# B&R Automation Studio project GroupProjectBR (part 3)

```iecst
			httpDecodeBase64_0();	// call FUB

			IF NOT(httpDecodeBase64_0.destLen=0) THEN
				Base64srcLen := httpDecodeBase64_0.destLen;
				httpDecodeBase64_0.enable := FALSE;
				ImageProcess := 0;
			END_IF;
	END_CASE;

END_PROGRAM

PROGRAM _EXIT
	(* Insert code here *)

END_PROGRAM
```

### Program Logical/Programs/Alarms (IEC)

#### Variables.var
```iecst
VAR
	test_alarm : BOOL;
	MpAlarmXCore_0 : MpAlarmXCore;
	pendingAlarms : BOOL;
	enableRedIcon : BOOL;
	enableYellowIcon : BOOL;
	redIconTimer : TON;
	timerCycle : BOOL;
	MpAlarmXHistory_0 : MpAlarmXHistory;
	MpUserXConfigType_0 : MpUserXConfigType;
	MpUserXConfig_0 : MpUserXConfig;
	isAcknowledged : BOOL;
	IsSemiAutoMode : BOOL;
	IsManualMode : BOOL;
END_VAR
```

#### Main.st
```iecst
PROGRAM _INIT
	(* Insert code here *)

END_PROGRAM

PROGRAM _CYCLIC
	(* Insert code here *)
	MpAlarmXCore_0.Enable := TRUE;
	MpAlarmXCore_0.MpLink := ADR(gAlarmXCore);
	MpAlarmXCore_0();

	MpAlarmXHistory_0.Enable := TRUE;
	MpAlarmXHistory_0.MpLink := ADR(gAlarmXHistory);
	MpAlarmXHistory_0();

	MpUserXConfig_0.Enable := TRUE;
	MpUserXConfig_0.Configuration := ADR(MpUserXConfigType_0);
	MpUserXConfig_0();

	redIconTimer.PT := T#500ms;
	redIconTimer();

	// HARDWARE ALARM DETECTION
	IF NOT ModuleOkActuators OR NOT ModuleOkCamera OR NOT ModuleOkEncoder OR NOT ModuleOkInverter OR NOT ModuleOkPLC_PLK OR NOT ModuleOkPneu_X67BC OR NOT ModuleOkScale THEN
		gAlarmHardware := TRUE;
	ELSE
		gAlarmHardware := FALSE;
	END_IF;

	//isAcknowledged := MpAlarmXCheckState(gAlarmXCore, 'test_alarm', mpALARMX_STATE_ACKNOWLEDGED);
	IF (MpAlarmXCheckState(gAlarmXCore, 'Unrecognized object', mpALARMX_STATE_ACKNOWLEDGED) AND
		MpAlarmXCheckState(gAlarmXCore, 'Left box is full', mpALARMX_STATE_ACKNOWLEDGED) AND
		MpAlarmXCheckState(gAlarmXCore, 'Hardware error', mpALARMX_STATE_ACKNOWLEDGED) AND
		MpAlarmXCheckState(gAlarmXCore, 'Motor error', mpALARMX_STATE_ACKNOWLEDGED) AND
		MpAlarmXCheckState(gAlarmXCore, 'Right box is full', mpALARMX_STATE_ACKNOWLEDGED)) THEN
		isAcknowledged := TRUE;
	ELSE
		isAcknowledged := FALSE;
	END_IF;

	IF (MpAlarmXCore_0.PendingAlarms > 0) THEN
		pendingAlarms := TRUE;
	ELSE
		pendingAlarms := FALSE;
	END_IF;

	IF (MpAlarmXCore_0.ActiveAlarms = 0 AND MpAlarmXCore_0.PendingAlarms > 0) THEN
		enableYellowIcon := TRUE;
	ELSE
		enableYellowIcon := FALSE;
	END_IF;

	IF (MpAlarmXCore_0.ActiveAlarms > 0) THEN
		gAlarmExist := TRUE;
		IF (NOT(isAcknowledged)) THEN
			//blinking
			IF (redIconTimer.IN = FALSE) THEN
				redIconTimer.IN := TRUE;
			ELSIF (redIconTimer.Q) THEN
				timerCycle := NOT timerCycle;
				redIconTimer.IN := FALSE;
			END_IF;
			enableRedIcon := timerCycle;
		ELSE
			//static
			enableRedIcon := TRUE;
		END_IF;
	ELSE
		gAlarmExist := FALSE;
		enableRedIcon := FALSE;
	END_IF;

END_PROGRAM

PROGRAM _EXIT
	(* Insert code here *)

END_PROGRAM
```

### Program Logical/Programs/PustyProgram

#### Main.st
```iecst
PROGRAM _INIT

END_PROGRAM

PROGRAM _CYCLIC

END_PROGRAM

PROGRAM _EXIT
	(* Insert code here *)

END_PROGRAM
```

### Program Logical/Programs/SemiAuto

#### Variables.var
```iecst
VAR
	Approval : BOOL;
	ActuatorByte : INT := 2#0000000000000000;
	ActuatorNotPushing : BOOL;
	ActuatorNotSorting : BOOL;
	ActuatorPushing : BOOL := FALSE;
	ActuatorSorting : BOOL := FALSE;
END_VAR
VAR CONSTANT
	ACTUATOR_BYTE_NOT_ACTIV : USINT := 2#0000000000000000;
	ACTUATOR_BYTE_PUSH : INT := 2#0000000000000100;
	ACTUATOR_BYTE_SORT : INT := 2#0000000000000001;
END_VAR
VAR
	AddToLeft : BOOL;
	AddToRight : BOOL;
	CTU_QuantityLeft : CTU;
	CTU_QuantityRight : CTU;
	CTU_Reset_Left : BOOL := FALSE;
	CTU_Reset_Right : BOOL;
	IsEnglishSelected : BOOL := TRUE;
	ItemDetected : BOOL := FALSE;
	ItemWeight : USINT;
	ItemWeightMeasured : USINT;
	MotorHome : BOOL;
	MotorInPosition : BOOL;
	MotorMoveAbsolute : BOOL := FALSE;
	MotorMoveDone : BOOL;
	MotorPos : LREAL;
	MotorPower : BOOL := FALSE;
	MotorReqAcc : UINT := 700;
	MotorReqDec : UINT := 700;
	MotorReqPosition : UINT := 0;
	MotorReqVel : {REDUND_UNREPLICABLE} UINT := 300;
	MotorResetError : BOOL := FALSE;
	MotorVel : REAL;
END_VAR
VAR CONSTANT
	MOTOR_DIST_LEFT : UINT := 90;
	MOTOR_DIST_RIGHT : UINT := 320;
END_VAR
VAR
	QuantityLeftStorage : UINT;
	QuantityRightStorage : UINT;
END_VAR
VAR CONSTANT
	RESET_ITEM_MEM_WEIGHT : USINT := 0;
END_VAR
VAR
	Start : BOOL := FALSE;
	State : ProgramStatesEnum := STOP;
	Stop : BOOL := FALSE;
	StringRecognisedModel : STRING[80];
	StringState : STRING[80];
	TimerActuatorOut : BOOL;
	TimerAfterDetect : BOOL;
	TimerCameraPicDone : BOOL;
	TimerTonActuator : TON;
	TimerTonActuatorIn : BOOL := FALSE;
	TimerTonCamera : TON;
	TimerTonDetect : TON;
END_VAR
VAR CONSTANT
	TIME_TON_ACTUATOR : TIME := T#500MS;
	TIME_TON_CAMERA : TIME := T#4S;
END_VAR
VAR
	TIME_TON_DETECT : TIME := T#2S;
	SemiAutoModeSelected : BOOL;
END_VAR
```

#### Main.st
```iecst
// ALREADY WORKING
PROGRAM _INIT
	// NEED ONLY FOR WATCH
	gAxis_1;
	gMotorBeltParType;
	gMotorBeltAxisBasic;
END_PROGRAM

PROGRAM _CYCLIC
	//CODE WORKS ONLY WHEN MANUAL MODE IS OFF
	SemiAutoModeSelected := (gMode=2);
	IF  SemiAutoModeSelected THEN
		// MOTOR MANAGEMENT
		gMotorBeltAxisBasic.Enable 		:= TRUE;
		gMotorBeltAxisBasic.MpLink 		:= ADR(gAxis_1);
		gMotorBeltAxisBasic.Parameters 	:= ADR(gMotorBeltParType);
		MotorMoveDone 					:= gMotorBeltAxisBasic.MoveDone;
		gMotorBeltAxisBasic.Power 		:= MotorPower;
		gMotorBeltAxisBasic.Home 		:= MotorHome;

		// IN STATE STOP VALUES DOESN'T FLUCTUATE
		IF gMotorBeltAxisBasic.Velocity > 15 THEN
			MotorVel := gMotorBeltAxisBasic.Velocity;
		ELSE
			MotorVel := 0;
		END_IF;
		IF gMotorBeltAxisBasic.Position > 5 THEN
			MotorPos := gMotorBeltAxisBasic.Position;
		ELSE
			MotorPos := 0;
		END_IF;

		// ASSIGNING MOTION PARAMETERS
		gMotorBeltParType.Acceleration 	:= MotorReqAcc;
		gMotorBeltParType.Deceleration 	:= MotorReqDec;
		gMotorBeltParType.Velocity 		:= MotorReqVel;
		gMotorBeltParType.Position 		:= MotorReqPosition;

		gMotorBeltAxisBasic();

		// ASSIGNING GLOBAL VARIABLES TO LOCAL VARIABLES
		gActuatorByte					 := ActuatorByte;
		gMotorBeltAxisBasic.Power 		 := MotorPower;
		gMotorBeltAxisBasic.MoveAbsolute := MotorMoveAbsolute;
		gMotorBeltAxisBasic.ErrorReset	 := MotorResetError;
		gStopState 						 := (State = 0);

		// ASSIGNING LOCAL VARIABLES TO GLOBAL VARIABLES
		MotorInPosition 				 := gMotorBeltAxisBasic.InPosition;
		ItemWeight 						 := gInWeightMeasure;

		// ITEM DETECTION CONDITION
		ItemDetected := (ItemWeight > 1);
		gWeightDetected := ItemDetected;

		// TIMERS
		// actuator
		TimerTonActuator(IN := TimerTonActuatorIn, PT := TIME_TON_ACTUATOR);
		TimerActuatorOut := TimerTonActuator.Q;
		// camera
		TimerTonCamera(IN := gImageAcq , PT := TIME_TON_CAMERA);
		TimerCameraPicDone := TimerTonCamera.Q;
		// delay after detection
		TimerTonDetect.IN := ItemDetected;
		TimerTonDetect.PT := TIME_TON_DETECT;
		TimerAfterDetect := TimerTonDetect.Q;
		TimerTonDetect();

		// COUNTERS - PRZENIESIONY NA SZYBKO DO AUTO

	END_IF;

	// ALARM OR STOP OR MANUAL TURNED ON
	IF	gAlarmHardware THEN	//ALARM
		IF NOT (State = ERROR) THEN
			State := ERROR;
		END_IF;
	ELSIF Stop OR NOT SemiAutoModeSelected OR gAlarmExist THEN
		Stop := FALSE;
		State := STOP;
	END_IF;

	// PROGRAM AUTO
	CASE State OF
		STOP:
			IF SemiAutoModeSelected THEN
				MotorPower 		  := FALSE;
				MotorMoveAbsolute := FALSE;
				MotorHome 		  := FALSE;
				MotorResetError   := FALSE;
			END_IF;
			MotorPos := 0;
			MotorVel := 0;
			StringState := 'Stop';
			TimerTonActuatorIn 	  := FALSE;
			ActuatorSorting 	  := FALSE;
			ActuatorPushing  	  := FALSE;
			IF Start THEN
				State := INIT;
			END_IF;

		INIT:
			StringState 		:= 'Inicjalizacja';
			ItemWeightMeasured 	:= RESET_ITEM_MEM_WEIGHT;
			gAddToRight 		:= FALSE;
			gAddToLeft 			:= FALSE;
			TimerTonActuatorIn 	:= FALSE;
			ActuatorSorting 	:= FALSE;
			ActuatorPushing 	:= FALSE;
			MotorMoveAbsolute 	:= FALSE;
			MotorPower 			:= TRUE;
			MotorHome 			:= TRUE;
			gPicNotRecognised	:= FALSE;
			State 				:= START;

		START:
			StringState 		:= 'Gotowy do startu';
			IF (ItemDetected AND Approval) THEN
				Approval := 0;
				State := DETECTION;
			END_IF;

		DETECTION:
			MotorHome 	:= FALSE;
			StringState := 'Wykrycie detalu';
			IF TimerAfterDetect THEN
				ItemWeightMeasured := ItemWeight;
				State := CATEGORIZATION;
			END_IF;

		CATEGORIZATION:
			StringState := 'Kategoryzacja detalu';
			IF gSorting.SortChoice = WEIGHT THEN
				State := DROP;
			ELSIF gSorting.SortChoice = OPTIC THEN
				State := TAKE_PICT_CAMERA;
			END_IF;

		TAKE_PICT_CAMERA:
			StringState := 'Robienie zdjecia';
			gImageAcq 	:= TRUE;
			IF TimerCameraPicDone AND Approval THEN
				StringState := 'Zdjecie zrobione';
				gDisplayImg := TRUE;
				Approval := 0;
				IF gSorting.RecognisedModel = 0 THEN 						//0
					gImageAcq 			  := FALSE;
					StringRecognisedModel := 'Unrecognised';
					State 				  := UNRECOGNISED_PIC;
				ELSE
					State 				  := DROP;
				END_IF;
			END_IF;

		DROP:
			StringState := 'Dozowanie detalu';
			ActuatorPushing := TRUE;
			IF TimerActuatorOut THEN
				ActuatorPushing := FALSE;
				IF gSorting.SortChoice = OPTIC THEN
					gSortChoiceView := TRUE;
					State := SORT_OPTIC;
				ELSIF gSorting.SortChoice = WEIGHT THEN
					gSortChoiceView := FALSE;
					State := SORT_WEIGHT;
				END_IF;
			END_IF;

		// ABOVE 1 TO ItemWeightChoosen ITEM FALL INTO THE LEFT, EQUAL AND ABOVE ItemWeightChoosen INTO THE RIGHT
		SORT_WEIGHT:
			StringState := 'Sortowanie wagowe';
			IF ItemWeightMeasured > 1 AND ItemWeightMeasured < gSorting.ItemWeightChoosen AND Approval THEN
				IF gSorting.SortLeftMin THEN
					Approval := 0;
					State := GO_STORAGE_LEFT;
				ELSE
					Approval := 0;
					State := GO_STORAGE_RIGHT;
				END_IF;
			ELSIF ItemWeightMeasured >= gSorting.ItemWeightChoosen AND Approval THEN
				IF gSorting.SortLeftMin THEN
					Approval := 0;
					State := GO_STORAGE_RIGHT;
				ELSE
					Approval := 0;
					State := GO_STORAGE_LEFT;
				END_IF;
			END_IF;

		SORT_OPTIC:
			StringState := 'Sortowanie optyczne';
			IF gSorting.RecognisedModel = 1 THEN
				gImageAcq 			  := FALSE;
				StringRecognisedModel := 'B&R';					//1
				IF gSorting.SortLeftBR AND Approval THEN
					Approval := 0;
					State := GO_STORAGE_LEFT;
				ELSE
					IF Approval THEN
						Approval := 0;
						State := GO_STORAGE_RIGHT;
					END_IF;
				END_IF;

			ELSIF gSorting.RecognisedModel = 2 THEN						//2
				gImageAcq 			  := FALSE;
				StringRecognisedModel := 'AS';
				IF gSorting.SortLeftBR AND Approval THEN
					Approval := 0;
					State := GO_STORAGE_RIGHT;
				ELSE
					IF Approval THEN
						Approval := 0;
						State := GO_STORAGE_LEFT;
					END_IF;
				END_IF;
			END_IF;

		GO_STORAGE_LEFT:
			StringState := 'Transport detalu do lewego zbiornika';
			MotorReqPosition := MOTOR_DIST_LEFT;
			MotorMoveAbsolute := TRUE;
			IF MotorInPosition AND MotorMoveDone AND Approval THEN
				Approval := 0;
				State := SORT_STORAGE_LEFT;
			END_IF;

		GO_STORAGE_RIGHT:
			StringState := 'Transport detalu do prawego zbiornika';
			MotorReqPosition  := MOTOR_DIST_RIGHT;
			MotorMoveAbsolute := TRUE;
			IF MotorInPosition AND MotorMoveDone AND Approval THEN
				Approval := 0;
				State := SORT_STORAGE_RIGHT;
			END_IF;

		SORT_STORAGE_LEFT:
			StringState := 'Zepchniecie detalu z tasmy do zbiornika lewego';
			MotorMoveAbsolute := FALSE;
			ActuatorSorting   := TRUE;
			gAddToLeft 		  := TRUE;
			IF TimerActuatorOut THEN
				State := INIT;
			END_IF;

		SORT_STORAGE_RIGHT:
			gAddToRight := TRUE;
			MotorMoveAbsolute := FALSE;
			State := INIT;

		UNRECOGNISED_PIC:
			StringState := 'Nie rozpoznano zdjecia';
			gPicNotRecognised := TRUE;
			State := STOP;

		ERROR:
			StringState := 'Wystapil blad';
			gErrorState := TRUE;
			IF gAlarmHardAck THEN
				IF NOT gAlarmHardware THEN
					gAlarmHardAck := FALSE;
					gErrorState := FALSE;
					State := STOP;
				END_IF;
			END_IF;

	END_CASE;

	// TIMER INPUT TRIGGER TO DELAY ACTUATORS
	IF ActuatorPushing OR ActuatorSorting THEN
		TimerTonActuatorIn := TRUE;
	ELSE
		TimerTonActuatorIn := FALSE;
	END_IF;

	// OPERATION OF BYTE ACTUATORS WITH TIMER
	IF ActuatorPushing THEN
		ActuatorByte := ACTUATOR_BYTE_PUSH;
		IF TimerActuatorOut THEN
			ActuatorPushing := FALSE;
		END_IF;
	ELSIF ActuatorSorting THEN
		ActuatorByte := ACTUATOR_BYTE_SORT;
		IF TimerActuatorOut THEN
			ActuatorSorting := FALSE;
		END_IF;
	ELSE
		ActuatorByte := ACTUATOR_BYTE_NOT_ACTIV;
	END_IF;

	// HMI GUYS WANTED SOME VARIABLES
	IF gSorting.SortChoice = OPTIC THEN
		gSortChoiceView := TRUE;
	ELSIF gSorting.SortChoice = WEIGHT THEN
		gSortChoiceView := FALSE;
	END_IF;

	ActuatorNotSorting := NOT ActuatorSorting;
	ActuatorNotPushing 	:= NOT ActuatorPushing;

	IF Start THEN
		Start := FALSE;
	END_IF;

	//Added by Jakub; Responsibler for changing machine state between English and Polish
	IF IsEnglishSelected THEN
		IF StringState = 'Inicjalizacja' THEN
			StringState := 'Initialization';

		ELSIF StringState = 'Zdjecie zrobione' THEN
			StringState := 'Picture taken';

		ELSIF StringState = 'Gotowy do startu' THEN
			StringState := 'Ready';

		ELSIF StringState = 'Wykrycie detalu' THEN
			StringState := 'Item detection';

		ELSIF StringState = 'Kategoryzacja detalu' THEN
			StringState := 'Item categorization';

		ELSIF StringState = 'Robienie zdjecia' THEN
			StringState := 'Taking a picture';

		ELSIF StringState = 'Dozowanie detalu' THEN
			StringState := 'Item dosing';

		ELSIF StringState = 'Sortowanie wagowe' THEN
			StringState := 'Sorting by weight';

		ELSIF StringState = 'Sortowanie optyczne' THEN
			StringState := 'Optical sorting';

		ELSIF StringState = 'Transport detalu do lewego zbiornika' THEN
			StringState := 'Item transport to the left tank';

		ELSIF StringState = 'Transport detalu do prawego zbiornika' THEN
			StringState := 'Item transport to the right tank';

		ELSIF StringState = 'Zepchniecie detalu z tasmy do zbiornika lewego' THEN
			StringState := 'Pushing the item from the belt to the left tank';

		ELSIF StringState = 'Nie rozpoznano zdjecia' THEN
			StringState := 'Photo not recognized';

		ELSIF StringState = 'Stop' THEN
			StringState := 'Stop';

		ELSIF StringState = 'Wystapil blad' THEN
			StringState := 'Error';

		ELSIF StringState = 'Gotowy do startu' THEN
			StringState := 'Ready to start';
		END_IF;
	END_IF;

		END_PROGRAM

PROGRAM _EXIT

		END_PROGRAM
```

### Program Logical/Programs/VisionCtr

#### Main.st
```iecst
PROGRAM _INIT
	gMotorBeltAxisBasic;
	gMotorBeltParType;
END_PROGRAM

PROGRAM _CYCLIC

	gAxis_1;
	gMotorBeltParType;
	gMotorBeltAxisBasic.MpLink := ADR(gAxis_1);
	gMotorBeltAxisBasic.Enable := TRUE;
	gMotorBeltAxisBasic.Parameters := ADR(gMotorBeltParType);
	//przypisywanie parametrów ruchu
	//	gMotorBeltParType.Direction := FORWARD;
	gMotorBeltParType.Acceleration := gMotorAcc;
	gMotorBeltParType.Deceleration := gMotorDec;
	gMotorBeltParType.Velocity := gMotorVel;
	gMotorBeltParType.Distance := gMotorDist;
	gMotorBeltAxisBasic();

END_PROGRAM

PROGRAM _EXIT
	(* Insert code here *)

END_PROGRAM
```

### Program Logical/Camera (IEC)

#### Variables.var
```iecst
VAR
	ImageAcqReady : BOOL;
	ImageAcqActive : BOOL;
	ImageAcq : BOOL;
	PhotosTaken : USINT;
	SET_FOCUS : UINT := 15000;
	MatchEnable : BOOL;
	NUM_SEARCH_MAX : USINT := 1;
	NumberMatches : USINT;
	EXPO_TIME : UDINT := 15000;
	FLASH_COLOR : USINT := 1;
	FLASH_SEGMENT : USINT := 0001;
	RecognisedModel : USINT;
	MIN_SCORE : USINT := 50;
	MAX_OVERLAP : USINT := 60;
END_VAR
```

#### Main.st
```iecst
PROGRAM _INIT
	(* Insert code here *)

	ImageAcqReady;
	ImageAcqActive;
	ImageAcq;
	PhotosTaken;
	NumberMatches;
	RecognisedModel;
	MatchEnable;

END_PROGRAM

PROGRAM _CYCLIC
	(* Insert code here *)

	gRecognisedModel := RecognisedModel;

END_PROGRAM

PROGRAM _EXIT
	(* Insert code here *)

END_PROGRAM
```

### Program Logical/Alarms (IEC)

#### Variables.var
```iecst
VAR
	test_alarm : BOOL;
	MpAlarmXCore_0 : MpAlarmXCore;
	pendingAlarms : BOOL;
  enableRedIcon : BOOL;
	enableYellowIcon : BOOL;
	redIconTimer : TON;
	timerCycle : BOOL;
	MpAlarmXHistory_0 : MpAlarmXHistory;
	isAcknowledged : BOOL;
  IsSemiAutoMode : BOOL;
	IsManualMode : BOOL;
END_VAR
```

#### Main.st
```iecst
PROGRAM _INIT
	(* Insert code here *)

END_PROGRAM

PROGRAM _CYCLIC
	(* Insert code here *)
	MpAlarmXCore_0.Enable := TRUE;
	MpAlarmXCore_0.MpLink := ADR(gAlarmXCore);
	MpAlarmXCore_0();

	MpAlarmXHistory_0.Enable := TRUE;
	MpAlarmXHistory_0.MpLink := ADR(gAlarmXHistory);
	MpAlarmXHistory_0();

	redIconTimer.PT := T#500ms;
	redIconTimer();

	isAcknowledged := MpAlarmXCheckState(gAlarmXCore, 'test_alarm', mpALARMX_STATE_ACKNOWLEDGED);

	IF (MpAlarmXCore_0.PendingAlarms > 0) THEN
		pendingAlarms := TRUE;
	ELSE
		pendingAlarms := FALSE;
	END_IF;

	IF (MpAlarmXCore_0.ActiveAlarms = 0 AND MpAlarmXCore_0.PendingAlarms > 0) THEN
		enableYellowIcon := TRUE;
	ELSE
		enableYellowIcon := FALSE;
	END_IF;

	IF (MpAlarmXCore_0.ActiveAlarms > 0) THEN
		IF (NOT(isAcknowledged)) THEN
			//blinking
			IF (redIconTimer.IN = FALSE) THEN
				redIconTimer.IN := TRUE;
			ELSIF (redIconTimer.Q) THEN
				timerCycle := NOT timerCycle;
				redIconTimer.IN := FALSE;
			END_IF;
			enableRedIcon := timerCycle;
		ELSE
			//static
			enableRedIcon := TRUE;
		END_IF;
	ELSE
		enableRedIcon := FALSE;
	END_IF;

END_PROGRAM

PROGRAM _EXIT
	(* Insert code here *)

END_PROGRAM
```

### Variables.var
```iecst
VAR
	Wysun : BOOL;
	MotorBeltAxisBasic : MpAxisBasic;
	MotorBeltParType : MpAxisBasicParType;
	BAIT : UINT;
END_VAR
```

### Program Logical/ProgramAuto

#### Main.st
```iecst
PROGRAM _INIT

END_PROGRAM

PROGRAM _CYCLIC

	IF gStart THEN

	END_IF;

	//	IF Wysun THEN  //TESTOWANIE
	//		BAIT := 2#0000_0000_0000_0101;
	//	ELSE
	//		BAIT := 2#0000_0000_0000_0000;
	//	END_IF;
	//Fragment kodu odpowiedzialny za inicjalizację taśmy
	gAxis_1;
	MotorBeltAxisBasic.MpLink := ADR(gAxis_1);
	MotorBeltAxisBasic.Enable := TRUE;
	MotorBeltAxisBasic.Parameters := ADR(MotorBeltParType);
	MotorBeltAxisBasic();

END_PROGRAM

PROGRAM _EXIT

END_PROGRAM
```

### Program Logical/ProgramManual

#### Types.typ
```iecst
TYPE
	ProcessRecipe : 	STRUCT
		Dopisz_skladniki : BOOL;
	END_STRUCT;
END_TYPE
```

#### Variables.var
```iecst
VAR
	ProcessRecipe0 : ProcessRecipe := (RedSign:=FALSE,Int:=0,Widget:=10,BiR:=FALSE,RiB:=0);
	MpRecipeXml_0 : MpRecipeXml;
	MpRecipeRegPar_0 : MpRecipeRegPar;
	MpRecipeUI_0 : MpRecipeUI;
	UIConnect0 : MpRecipeUIConnectType;
END_VAR
```

#### Main.st
```iecst
PROGRAM _INIT

END_PROGRAM

PROGRAM _CYCLIC

END_PROGRAM

PROGRAM _EXIT

END_PROGRAM
```

### Program Logical/RecipeManag

#### Main.st
```iecst
PROGRAM _INIT
	MpRecipeRegPar_0(MpLink := ADR(gRecipeXml) , Enable := TRUE, PVName := ADR('ProgramManual:ProcessRecipe0')); //tutaj zmienna do edycji
	MpRecipeXml_0(MpLink := ADR(gRecipeXml), Enable := TRUE, DeviceName := ADR('CF'), FileName := ADR('Recipes'));
	MpRecipeUI_0(MpLink := ADR(gRecipeXml), Enable := TRUE, UIConnect := ADR(UIConnect0) );
END_PROGRAM

PROGRAM _CYCLIC
	//Pamiętaj pozmieniać strukturę wraz ze zmienna
	MpRecipeXml_0();
	MpRecipeRegPar_0();
	MpRecipeUI_0();
END_PROGRAM

PROGRAM _EXIT
	MpRecipeXml_0(Enable := FALSE);
	MpRecipeXml_0();

	MpRecipeRegPar_0(Enable := FALSE);
	MpRecipeRegPar_0();

	MpRecipeUI_0(Enable := FALSE);
	MpRecipeUI_0();
END_PROGRAM
```
